{attribute addProperty BoxType "EL2595-0000-0018"}
{attribute addProperty Id "StatusAT %I*Status_8453BAB9162"}
{attribute addProperty CRC "614162207"}
{attribute addProperty SizeInBites "16"}
{attribute addProperty SizeInBytes "2"}
TYPE DOX_Status_249B5F1F :
STRUCT
	{attribute addProperty Name "Status"}
	Status AT %I* : Status_8453BAB9;
END_STRUCT
END_TYPE

(* stored: Version 1.2.0.0, ProductVersion 3.1.4024.9
   DUT DOX_Status_249B5F1F: Id {d3c2e09d-2233-41b9-a9b5-acc0e5076e66} *)
